PROGRAM MAIN
VAR
END_VAR

END_PROGRAM

(* stored: Version 1.1.0.1
   POU MAIN: Id {cf4625e2-375c-47c1-b85d-d3fce8ed47d6} *)
